Omron Sysmac Studio project mixer_Recuperato (Sysmac Studio 1.56.0.11, StandardProject)

# Controller new_Controller_0: NX1P2-9024DT1 version 1.64
Task PrimaryTask (priority 4, period or condition 2000): Programma0

TYPE ricetta : STRUCT
    massimo : INT;
    minimo : INT;
END_STRUCT END_TYPE

VAR_GLOBAL
    ricetta1 : ricetta;
    array_ricette : ARRAY[0..2] OF ricetta;
    Sens_livello : INT := 0;  (* at IOBus://unit#1/Ch1 Analog Input Value *)
    svuotamento : BOOL;  (* at BuiltInIO://cpu/#0/Output_Bit_00 *)
    riempimento : BOOL;  (* at BuiltInIO://cpu/#0/Output_Bit_01 *)
    mot_mixer : BOOL;  (* at BuiltInIO://cpu/#0/Output_Bit_02 *)
    start : BOOL := False;  (* at BuiltInIO://cpu/#0/Input_Bit_00 *)
    ricetta_scelta : DINT;
    max_presonalizzato : INT;
    min_personalizzato : INT;
    curr_livello_min : DINT;
    curr_livello_max : DINT;
    fill_liquido : DINT;
END_VAR

PROGRAM Programma0
VAR
    stato : INT;
    array_ricette : ARRAY[0..2] OF ricetta := [(massimo := 80, minimo := 20), (massimo := 75, minimo := 10), (massimo := 0, minimo := 0)];
    timer_finito : BOOL;
    trigger_timer : BOOL;
    timer_lav : TON;
    timer_set : TIME;
END_VAR
VAR_EXTERNAL
    start : BOOL;
    svuotamento : BOOL;
    riempimento : BOOL;
    mot_mixer : BOOL;
    Sens_livello : INT;
    ricetta_scelta : DINT;
    max_presonalizzato : INT;
    min_personalizzato : INT;
    curr_livello_min : DINT;
    curr_livello_max : DINT;
END_VAR
CASE stato OF
	0://fermo
		Sens_livello := 0;
		svuotamento := FALSE;
		riempimento := FALSE;
		mot_mixer := FALSE;
		curr_livello_min :=  array_ricette[ricetta_scelta].minimo;
		curr_livello_max := array_ricette[ricetta_scelta].massimo;
		
			IF ricetta_scelta = 2 THEN
				 array_ricette[2].massimo := max_presonalizzato;
				 array_ricette[2].minimo := min_personalizzato;
			END_IF;
			
		IF start THEN
			stato := 1;
		END_IF;
		
		1://riempimento
			timer_set := T#500ms;
			svuotamento := FALSE;
			riempimento := TRUE;
			mot_mixer := FALSE;
			IF timer_finito THEN
				Sens_livello := Sens_livello + 1;
			END_IF;
			IF Sens_livello >= array_ricette[ricetta_scelta].massimo THEN
				stato := 2;
				timer_set := T#5s;
			END_IF;
		
		2://mix
			timer_set := T#5s;
			svuotamento := FALSE;
			riempimento := FALSE;
			mot_mixer := TRUE;
			IF timer_finito THEN
				stato := 3;
			END_IF;
	3://svuotamento
			timer_set := T#500ms;
			svuotamento := TRUE;
			riempimento := FALSE;
			mot_mixer := FALSE;
			IF timer_finito THEN
				Sens_livello := Sens_livello - 1;
			END_IF;
			IF Sens_livello <= array_ricette[ricetta_scelta].minimo THEN
				stato := 0;
			END_IF;
		END_CASE ;

timer_lav(In:=trigger_timer OR riempimento OR svuotamento , PT:=timer_set, Q=>timer_finito);
END_PROGRAM

# Device HMI_NA5_0 (NA): not converted